Fanuc KAREL source: kt00102.KL

-- PROVISIONAL review KL for V1013-1; original PC SHA256 2ab0b0f2a76e57a9287293cf257f200f3d99955c4b7d69d89afafc5106a375b7
-- Incomplete behavior may be omitted. Consult companion uncertainty JSON. Do not deploy.
PROGRAM KT00102
%NOLOCKGROUP
VAR
  I1 : INTEGER
  OUT : REAL
-- UNRESOLVED_DECL Y2 type=002018
BEGIN
  -- UNRESOLVED_PC offsets 5-16; opcodes 2E,23
  -- UNRESOLVED_PC offsets 21-35; opcodes 2E,22,9D,33,B2
  -- UNRESOLVED_PC offsets 40-66; opcodes 21,22,9D,33,B1,64,29,64,29,6C,23
  -- UNRESOLVED_PC offsets 71-75; opcodes 7F
END KT00102
